{attribute addProperty BoxType "EL2502-0010-0020"}
{attribute addProperty Id "SysTimeAT %I*ULINT648"}
{attribute addProperty CRC "3497641984"}
{attribute addProperty SizeInBites "64"}
{attribute addProperty SizeInBytes "8"}
TYPE PWM_SysTime_Channel_D079C800 :
STRUCT
	{attribute addProperty Name "SysTime"}
	SysTime AT %I* : ULINT;
END_STRUCT
END_TYPE

(* stored: Version 1.2.0.0, ProductVersion 3.1.4024.9
   DUT PWM_SysTime_Channel_D079C800: Id {11fa2753-27f1-4c52-a369-0056d5b5dcc6} *)
